FUNCTION_BLOCK FB_PIDR (* PID with Bumpless Transfer and Anti-Reset Windup, REAL PV+XOUT *)
  (* Standard: 61499-1-D.1 *)
  (* Version 0.4, 2010-12-18, JHC, Holobloc Inc, Updated REQ algorithm to one statement per line for new regexp ST/Java conversion. *)
  (* Version 0.3, 2010-12-03, JHC, Holobloc Inc, Corrected & regression tested anti-reset windup. *)
  (* Version 0.2, 2010-12-03, JHC, Holobloc Inc, Corrected & regression tested bumpless MANUAL/AUTO transfer. *)
  (* Version 0.1, 2010-12-03, JHC, Holobloc Inc, Made a SimpleFB. *)
  (* Version 0.0, 2004-09-06, JHC, Rockwell Automation *)
  (* Compiler header: package fb.rt.process; *)
  (* Compiler classdef: SimpleFB *)
  (* Compiler Java Sun JDK 1.6.0 *)
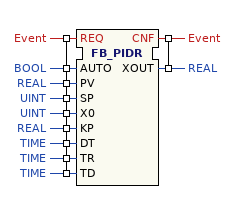
  EVENT_INPUT
    REQ WITH AUTO, PV, SP, X0, KP, TR, TD, DT;
  END_EVENT
  EVENT_OUTPUT
    CNF WITH XOUT;
  END_EVENT
  VAR_INPUT
    AUTO : BOOL; (* 0-manual,1-automatic *)
    PV : REAL; (* Process variable,0-100 percent *)
    SP : UINT; (* Set Point,0-100 percent *)
    X0 : UINT; (* Manual Output Setting,0-100 percent *)
    KP : REAL; (* Proportionality Constant *)
    DT : TIME := t#1s; (* Sampling Period *)
    TR : TIME; (* Reset Time *)
    TD : TIME; (* Derivative Time Constant *)
  END_VAR
  VAR_OUTPUT
    XOUT : REAL; (* Manipulated Variable,0-100 percent *)
  END_VAR
  VAR
    WASAUTO : BOOL;
    WASLIMITED : BOOL;
    ERROR : REAL;
    ITERM : REAL;
    DTERM : REAL;
    X1 : REAL;
    X2 : REAL;
    X3 : REAL;
  END_VAR
  ALGORITHM REQ IN ST:
ERROR:=PV-SP;
IF AUTO THEN
  IF WASAUTO AND NOT WASLIMITED THEN
    ITERM:=ITERM+ERROR*DT/TR;
    DTERM:=(3*(PV-X3)+X1-X2)*TD/DT/10;
  ELSE
    ITERM:=-KP*ERROR-XOUT;
    DTERM:=0;
  END_IF;
  XOUT:=-KP*ERROR-ITERM-DTERM;
ELSE XOUT:=X0;
END_IF
X3:=X2;
X2:=X1;
X1:=PV;
WASLIMITED := FALSE;
IF XOUT<0 THEN
  XOUT:=0;
  WASLIMITED := TRUE;
ELSIF XOUT>100 THEN
  XOUT:=100;
  WASLIMITED := TRUE;
END_IF;
WASAUTO:=AUTO;
  END_ALGORITHM
END_FUNCTION_BLOCK
